                        (* send frame *)
                        fbSend(bExecute  := FALSE);
                        fbSend(sSrvNetID := '',
                               hSocket   := fbConnect.hSocket,
                               cbLen     := SIZEOF(toServer.Header) + _byteCount,(* size of header + size of user data *)
                               pSrc      := ADR(toServer),(* pointer to the frame data *)
                               bExecute  := TRUE,
                               tTimeout  := T#5s);

                        tx_state := 1;
                    END_IF
                1:(* wait until send not busy *)
                    fbSend( bExecute := FALSE );
                    IF NOT fbSend.bBusy THEN
                        tx_state := 0;
                        IF NOT fbSend.bError THEN(* no error *)
                            ;
                        ELSE(* send error => log error and disconnect *)
                            errors.Error(nErrId := fbSend.nErrId );
                            bDisconnect := TRUE;(* set flag *)
                        END_IF
                    END_IF
            END_CASE

            (* ------------------------------------------- Get/fetch rx data ----------------------------------------------------------------- *)
            CASE rx_state OF
                0:
                    IF NOT bDisconnect THEN
                        pollTimer( IN := TRUE );
                        IF pollTimer.Q THEN
                            pollTimer( IN := FALSE );

                            fbReceive( bExecute := FALSE );
                            fbReceive( 	sSrvNetId	:= '',
                            hSocket		:= fbConnect.hSocket,
                            cbLen		:= SIZEOF(fromServer) - cbReceived,
                            pDest		:= ADR(fromServer) + cbReceived,
                            bExecute	:= TRUE,
                            tTimeout	:= T#5s );
                            rx_state := 1;
                        END_IF
                    END_IF
                1:(* wait until receive not busy *)
                    fbReceive( bExecute := FALSE );
                    IF NOT fbReceive.bBusy THEN
                        rx_state := 0;
                        IF NOT fbReceive.bError THEN
                            IF fbReceive.nRecBytes > 0 THEN (* some bytes received *)

                                pollTimer( PT := T#0s );(* increase polling speed *)
                                cbReceived := cbReceived + fbReceive.nRecBytes;

                                (* parse received bytes *)
                                REPEAT
                                    bAbort := TRUE;(* set flag *)
                                    IF cbReceived >= SIZEOF(fromServer.Header) THEN (* all header bytes received => check header data *)

                                        (* correct header data *)
                                        fromServer.Header.ByteCount    := BE32_TO_HOST(fromServer.Header.ByteCount);
                                        Counter                        := fromServer.Header.Counter;
                                        fromServer.Header.SentTime     := BE32_TO_HOST(fromServer.Header.SentTime);
                                        fromServer.Header.DatagramType := BE32_TO_HOST(fromServer.Header.DatagramType);

                                        IF (fromServer.Header.ByteCount <= SIZEOF( fromServer.Payload))(* check frame (user data) length *)
                                        THEN

                                            cbRx := SIZEOF(fromServer.Header) + fromServer.Header.ByteCount;(* calculate the (expected) length of the rx frame *)
                                            IF cbReceived >= cbRx  THEN (* all frame bytes received? *)

                                               (* currently only use the data on a 32 Bit raw image *)
                                                IF fromServer.Header.DatagramType = MNG_Raw32BitImage THEN

                                                    IF 48 = (fromServer.Header.ByteCount - 4) THEN

                                                        (* BOOL Cocktail_Holder1_00_VACUUM *)
                                                        Inputs.Cocktail_Holder1_00_VACUUM := fromServer.Payload[2]<>0;

                                                        (* BOOL DetectionCookieAdapter1_00_IR *)
                                                        Inputs.DetectionCookieAdapter1_00_IR := fromServer.Payload[3]<>0;

                                                        (* BOOL Cocktail_Holder2_00_VACUUM *)
                                                        Inputs.Cocktail_Holder2_00_VACUUM := fromServer.Payload[4]<>0;

                                                        (* BOOL DetectionCookieAdapter2_00_IR *)
                                                        Inputs.DetectionCookieAdapter2_00_IR := fromServer.Payload[5]<>0;

                                                        (* BOOL Cocktail_Holder3_00_VACUUM *)
                                                        Inputs.Cocktail_Holder3_00_VACUUM := fromServer.Payload[6]<>0;

                                                        (* BOOL DetectionCookieAdapter3_00_IR *)
                                                        Inputs.DetectionCookieAdapter3_00_IR := fromServer.Payload[7]<>0;

                                                        (* BOOL Cocktail_Holder4_00_VACUUM *)
                                                        Inputs.Cocktail_Holder4_00_VACUUM := fromServer.Payload[8]<>0;

                                                        (* BOOL DetectionCookieAdapter4_00_IR *)
                                                        Inputs.DetectionCookieAdapter4_00_IR := fromServer.Payload[9]<>0;

                                                        (* BOOL Cocktail_Holder5_00_VACUUM *)
                                                        Inputs.Cocktail_Holder5_00_VACUUM := fromServer.Payload[10]<>0;

                                                        (* BOOL DetectionCookieAdapter5_00_IR *)
                                                        Inputs.DetectionCookieAdapter5_00_IR := fromServer.Payload[11]<>0;

                                                        (* BOOL Cocktail_Holder6_00_VACUUM *)
                                                        Inputs.Cocktail_Holder6_00_VACUUM := fromServer.Payload[12]<>0;

                                                        (* BOOL DetectionCookieAdapter6_00_IR *)
                                                        Inputs.DetectionCookieAdapter6_00_IR := fromServer.Payload[13]<>0;

                                                    ELSE(* receive error: invalid frame format/data *)
                                                        errors.Error(nErrId := PLCPRJ_ERROR_INVALID_IO_FORMAT_RECEIVED );
                                                    END_IF

                                                END_IF

                                                MEMMOVE( ADR( fromServer ), ADR( fromServer ) + cbRx,  cbReceived - cbRx );(* shift the remaining rx bytes *)
                                                cbReceived := cbReceived - cbRx;(* recalculate the size of the remaining rx bytes *)

                                                bAbort := FALSE;(* reset flag, try to parse next frame *)

                                                (* ELSE repeat reading *)
                                            END_IF

                                        ELSE(* receive error: invalid frame format/data *)
                                            errors.Error(nErrId := PLCPRJ_ERROR_INVALID_FRAME_FORMAT );
                                            bDisconnect := TRUE;(* set flag *)
                                        END_IF
                                        (* ELSE repeat reading *)
                                    END_IF (* IF cbReceived >= SIZEOF(rxFrame.head) THEN *)

                                UNTIL bAbort
                                END_REPEAT

                            ELSE(* fbReceive.nRecBytes = 0, repeat reading *)
                                pollTimer( PT := PLCPRJ_RECEIVER_POLLING_CYCLE_TIME );(* slow down the polling cycle *)
                            END_IF(* IF fbReceive.nRecBytes > 0 THEN *)
                        ELSE(* receive error => log error and disconnect *)
                            errors.Error(nErrId := fbReceive.nErrId );
                            bDisconnect := TRUE;(* set flag *)
                        END_IF

                    END_IF(*IF NOT fbReceive.bBusy THEN*)

            END_CASE

        END_IF

    3:(* disconnect *)
        fbConnect( bEnable:= FALSE, eState=>eState );
        IF eState = eSOCKET_DISCONNECTED THEN
            state := 0;
        END_IF

END_CASE

END_FUNCTION_BLOCK

// ---- POUs/industrialPhysics/FB_LogFifo.TcPOU
/// Log/debug/error message fifo 
FUNCTION_BLOCK FB_LogFifo
VAR_INPUT
	/// TRUE => Enable log message output, FALSE => Disable 
	bLog: BOOL := FALSE;
	/// Log message description string (allows the identification of log message source) 
	sPrefix: STRING := 'Unknown::';
	/// String message to add (write) to the fifo 
	sMessage: STRING := '';
	/// Error code to add (write) to the fifo 
	nErrID: UDINT := 0;
	/// Socket connection handle 
	hSocket: T_HSOCKET;
END_VAR
VAR_OUTPUT
	/// TRUE = New entry added or removed succesfully, FALSE = Fifo overflow or fifo empty 
	bOk: BOOL;
	/// String entry removed (read) from fifo 
	sGet: T_MaxString := '';
	/// Number of fifo entries 
	nCount: UDINT := 0;
END_VAR
VAR
	/// Basic (lower level) string buffer control function block 
	fbBuffer: FB_StringRingBuffer;
	/// Internal buffer memory 
	buffer: ARRAY[0..PLCPRJ_BUFFER_SIZE] OF BYTE;
	sSource: T_MaxString;
	sPut: T_MaxString;
END_VAR

;

ACTION Remove:
(* Removes oldest fifo entry *)
IF nCount = 0 THEN
	sGet := '';
	bOk := FALSE;
	RETURN;
END_IF

fbBuffer.A_RemoveHead( pBuffer:= ADR(buffer), cbBuffer:= SIZEOF(buffer),
						getValue=>sGet, bOk=>bOk, nCount=>nCount );
END_ACTION

ACTION Message:
(* Adds new fifo entry *)
sPut := CONCAT( CONCAT( sPrefix, sMessage ), CONCAT( '::', HSOCKET_TO_STRING(hSocket) ) );
fbBuffer.A_AddTail( pBuffer:= ADR(buffer), cbBuffer:= SIZEOF(buffer),
					putValue:= sPut, bOk=>bOk, nCount=>nCount );
IF bOk THEN
	IF bLog THEN(* Log information message *)
		ADSLOGSTR( ADSLOG_MSGTYPE_HINT OR ADSLOG_MSGTYPE_LOG, '%s', sPut );	
	END_IF
END_IF
END_ACTION

ACTION Clear:
(* Clears all fifo entries *)
fbBuffer.A_Reset( 	pBuffer := ADR( buffer ), cbBuffer := SIZEOF( buffer ), 
					bOk=>bOk, nCount=>nCount, getValue=>sGet );
END_ACTION

ACTION Error:
(* Adds new fifo entry *)
IF nErrID = 0 THEN
	sSource := '::Error: 0x';
ELSIF ( nErrID AND 16#80000000) = 16#80000000 THEN
	IF nErrID = 16#80072746 THEN
		sSource := '::Win32 error (the connection is reset by remote side): 0x';
	ELSE
		sSource := '::Win32 error: 0x';
	END_IF
ELSIF (nErrID AND 16#00008100) = 16#00008100 THEN
	CASE nErrID OF
		PLCPRJ_ERROR_RECEIVE_TIMEOUT:
			sSource := '::PLC sample project receive timeout error: 0x';
		PLCPRJ_ERROR_SENDFIFO_OVERFLOW:
			sSource := '::PLC sample project send fifo overflow error: 0x';
		PLCPRJ_ERROR_RECFIFO_OVERFLOW:
			sSource := '::PLC sample project receive fifo overflow error: 0x';
		PLCPRJ_ERROR_INVALID_FRAME_FORMAT:
			sSource := '::PLC sample project invalid frame format error: 0x';
	ELSE
		sSource := '::Other PLC sample project error: 0x';
	END_CASE
ELSIF (nErrID AND 16#00008000) = 16#00008000 THEN
	sSource := '::Internal TCP/IP Connection Server error: 0x';
ELSE
	sSource := '::TwinCAT System error: 0x';
END_IF

sPut := CONCAT( CONCAT( CONCAT( sPrefix, sMessage ), sSource ), DWORD_TO_HEXSTR( nErrID AND 16#FFFF, 0, FALSE ) ); 

fbBuffer.A_AddTail( pBuffer:= ADR(buffer), cbBuffer:= SIZEOF(buffer),
					putValue:= sPut, bOk=>bOk, nCount=>nCount );
IF bOk THEN
	IF bLog THEN(* Log error message *)
		ADSLOGSTR( ADSLOG_MSGTYPE_ERROR OR ADSLOG_MSGTYPE_LOG, '%s', sPut );	
	END_IF
END_IF
END_ACTION

END_FUNCTION_BLOCK

// ---- POUs/industrialPhysics/FB_IOLink.TcPOU
FUNCTION_BLOCK FB_IOLink
VAR_INPUT
	goon : BOOL  := TRUE;
	inputs: MNG_Application_Inputs_32Bit;
	
	
END_VAR
VAR_OUTPUT
	outputs: MNG_Application_Outputs_32Bit;
END_VAR
VAR
	timer: ARRAY[1..6] OF Tc2_Standard.TON;
	state: ARRAY[1..6] OF INT := [0, 0, 0, 0, 0, 0];
	deltaMover: ARRAY[1..6] OF LREAL;
END_VAR

// Application code follows here:

IF goon THEN

outputs.Fahrachse1_00_ChainDrvActual := GVL.ax[1].NcToPlc.SetPos/1000;
outputs.Fahrachse2_00_ChainDrvActual := GVL.ax[2].NcToPlc.SetPos/1000;
outputs.Fahrachse3_00_ChainDrvActual := GVL.ax[3].NcToPlc.SetPos/1000;
outputs.Fahrachse4_00_ChainDrvActual := GVL.ax[4].NcToPlc.SetPos/1000;
outputs.Fahrachse5_00_ChainDrvActual := GVL.ax[5].NcToPlc.SetPos/1000;
outputs.Fahrachse6_00_ChainDrvActual := GVL.ax[6].NcToPlc.SetPos/1000;


outputs.LED_0_00_00_on1 := GVL.LampInterface[1][1];
outputs.LED_0_05_00_on1 := GVL.LampInterface[1][2];
outputs.LED_0_10_00_on1 := GVL.LampInterface[1][3];
outputs.LED_0_15_00_on1 := GVL.LampInterface[1][4];
outputs.LED_0_20_00_on1 := GVL.LampInterface[1][5];
outputs.LED_0_25_00_on1 := GVL.LampInterface[1][6];
outputs.LED_0_30_00_on1 := GVL.LampInterface[1][7];
outputs.LED_0_35_00_on1 := GVL.LampInterface[1][8];
outputs.LED_0_40_00_on1 := GVL.LampInterface[1][9];
outputs.LED_0_45_00_on1 := GVL.LampInterface[1][10];
outputs.LED_0_50_00_on1 := GVL.LampInterface[1][11];
outputs.LED_0_55_00_on1 := GVL.LampInterface[1][12];
outputs.LED_0_60_00_on1 := GVL.LampInterface[1][13];
outputs.LED_0_65_00_on1 := GVL.LampInterface[1][14];
outputs.LED_0_70_00_on1 := GVL.LampInterface[1][15];
outputs.LED_0_75_00_on1 := GVL.LampInterface[1][16];
outputs.LED_0_80_00_on1 := GVL.LampInterface[1][17];
outputs.LED_0_85_00_on1 := GVL.LampInterface[1][18];
outputs.LED_0_90_00_on1 := GVL.LampInterface[1][19];
outputs.LED_0_95_00_on1 := GVL.LampInterface[1][20];
outputs.LED_1_00_00_on1 := GVL.LampInterface[1][21];
outputs.LED_1_05_00_on1 := GVL.LampInterface[1][22];
outputs.LED_1_10_00_on1 := GVL.LampInterface[1][23];
outputs.LED_1_15_00_on1 := GVL.LampInterface[1][24];
outputs.LED_1_20_00_on1 := GVL.LampInterface[1][25];
outputs.LED_1_25_00_on1 := GVL.LampInterface[1][26];
outputs.LED_1_30_00_on1 := GVL.LampInterface[1][27];
outputs.LED_1_35_00_on1 := GVL.LampInterface[1][28];
outputs.LED_1_40_00_on1 := GVL.LampInterface[1][29];
outputs.LED_1_45_00_on1 := GVL.LampInterface[1][30];
(*
outputs.LED_1_50_00_on1 := GVL.LampInterface[1][31];
outputs.LED_1_55_00_on1 := GVL.LampInterface[1][32];
outputs.LED_1_60_00_on1 := GVL.LampInterface[1][33];
outputs.LED_1_65_00_on1 := GVL.LampInterface[1][34];
outputs.LED_1_70_00_on1 := GVL.LampInterface[1][35];
outputs.LED_1_75_00_on1 := GVL.LampInterface[1][36];
outputs.LED_1_80_00_on1 := GVL.LampInterface[1][37];
outputs.LED_1_85_00_on1 := GVL.LampInterface[1][38];
outputs.LED_1_90_00_on1 := GVL.LampInterface[1][39];
outputs.LED_1_95_00_on1 := GVL.LampInterface[1][40];
*)
outputs.LED_2_00_00_on1 := GVL.LampInterface[1][41];
outputs.LED_2_05_00_on1 := GVL.LampInterface[1][42];
outputs.LED_2_10_00_on1 := GVL.LampInterface[1][43];
outputs.LED_2_15_00_on1 := GVL.LampInterface[1][44];
outputs.LED_2_20_00_on1 := GVL.LampInterface[1][45];
outputs.LED_2_25_00_on1 := GVL.LampInterface[1][46];
outputs.LED_2_30_00_on1 := GVL.LampInterface[1][47];
outputs.LED_2_35_00_on1 := GVL.LampInterface[1][48];
outputs.LED_2_40_00_on1 := GVL.LampInterface[1][49];
outputs.LED_2_45_00_on1 := GVL.LampInterface[1][50];
outputs.LED_2_50_00_on1 := GVL.LampInterface[1][51];
outputs.LED_2_55_00_on1 := GVL.LampInterface[1][52];
outputs.LED_2_60_00_on1 := GVL.LampInterface[1][53];
outputs.LED_2_65_00_on1 := GVL.LampInterface[1][54];
outputs.LED_2_70_00_on1 := GVL.LampInterface[1][55];
outputs.LED_2_75_00_on1 := GVL.LampInterface[1][56];
outputs.LED_2_80_00_on1 := GVL.LampInterface[1][57];
outputs.LED_2_85_00_on1 := GVL.LampInterface[1][58];
outputs.LED_2_90_00_on1 := GVL.LampInterface[1][59];
outputs.LED_2_95_00_on1 := GVL.LampInterface[1][60];
outputs.LED_3_00_00_on1 := GVL.LampInterface[1][61];
outputs.LED_3_05_00_on1 := GVL.LampInterface[1][62];
outputs.LED_3_10_00_on1 := GVL.LampInterface[1][63];
outputs.LED_3_15_00_on1 := GVL.LampInterface[1][64];
outputs.LED_3_20_00_on1 := GVL.LampInterface[1][65];
outputs.LED_3_25_00_on1 := GVL.LampInterface[1][66];
outputs.LED_3_30_00_on1 := GVL.LampInterface[1][67];
outputs.LED_3_35_00_on1 := GVL.LampInterface[1][68];
outputs.LED_3_40_00_on1 := GVL.LampInterface[1][69];
outputs.LED_3_45_00_on1 := GVL.LampInterface[1][70];
(*
outputs.LED_3_50_00_on1 := GVL.LampInterface[1][71];
outputs.LED_3_55_00_on1 := GVL.LampInterface[1][72];
outputs.LED_3_60_00_on1 := GVL.LampInterface[1][73];
outputs.LED_3_65_00_on1 := GVL.LampInterface[1][74];
outputs.LED_3_70_00_on1 := GVL.LampInterface[1][75];
outputs.LED_3_75_00_on1 := GVL.LampInterface[1][76];
outputs.LED_3_80_00_on1 := GVL.LampInterface[1][77];
outputs.LED_3_85_00_on1 := GVL.LampInterface[1][78];
outputs.LED_3_90_00_on1 := GVL.LampInterface[1][79];
outputs.LED_3_95_00_on1 := GVL.LampInterface[1][80];
*)

// Lampe 2:

outputs.LED_0_00_00_on2 := GVL.LampInterface[2][1];;
outputs.LED_0_05_00_on2 := GVL.LampInterface[2][2];;
outputs.LED_0_10_00_on2 := GVL.LampInterface[2][3];;
outputs.LED_0_15_00_on2 := GVL.LampInterface[2][4];;
outputs.LED_0_20_00_on2 := GVL.LampInterface[2][5];;
outputs.LED_0_25_00_on2 := GVL.LampInterface[2][6];;
outputs.LED_0_30_00_on2 := GVL.LampInterface[2][7];;
outputs.LED_0_35_00_on2 := GVL.LampInterface[2][8];;
outputs.LED_0_40_00_on2 := GVL.LampInterface[2][9];;
outputs.LED_0_45_00_on2 := GVL.LampInterface[2][10];
outputs.LED_0_50_00_on2 := GVL.LampInterface[2][11];
outputs.LED_0_55_00_on2 := GVL.LampInterface[2][12];
outputs.LED_0_60_00_on2 := GVL.LampInterface[2][13];
outputs.LED_0_65_00_on2 := GVL.LampInterface[2][14];
outputs.LED_0_70_00_on2 := GVL.LampInterface[2][15];
outputs.LED_0_75_00_on2 := GVL.LampInterface[2][16];
outputs.LED_0_80_00_on2 := GVL.LampInterface[2][17];
outputs.LED_0_85_00_on2 := GVL.LampInterface[2][18];
outputs.LED_0_90_00_on2 := GVL.LampInterface[2][19];
outputs.LED_0_95_00_on2 := GVL.LampInterface[2][20];
outputs.LED_1_00_00_on2 := GVL.LampInterface[2][21];
outputs.LED_1_05_00_on2 := GVL.LampInterface[2][22];
outputs.LED_1_10_00_on2 := GVL.LampInterface[2][23];
outputs.LED_1_15_00_on2 := GVL.LampInterface[2][24];
outputs.LED_1_20_00_on2 := GVL.LampInterface[2][25];
outputs.LED_1_25_00_on2 := GVL.LampInterface[2][26];
outputs.LED_1_30_00_on2 := GVL.LampInterface[2][27];
outputs.LED_1_35_00_on2 := GVL.LampInterface[2][28];
outputs.LED_1_40_00_on2 := GVL.LampInterface[2][29];
outputs.LED_1_45_00_on2 := GVL.LampInterface[2][30];
(*                                                 
outputs.LED_1_50_00_on2 := GVL.LampInterface[2][31];
outputs.LED_1_55_00_on2 := GVL.LampInterface[2][32];
outputs.LED_1_60_00_on2 := GVL.LampInterface[2][33];
outputs.LED_1_65_00_on2 := GVL.LampInterface[2][34];
outputs.LED_1_70_00_on2 := GVL.LampInterface[2][35];
outputs.LED_1_75_00_on2 := GVL.LampInterface[2][36];
outputs.LED_1_80_00_on2 := GVL.LampInterface[2][37];
outputs.LED_1_85_00_on2 := GVL.LampInterface[2][38];
outputs.LED_1_90_00_on2 := GVL.LampInterface[2][39];
outputs.LED_1_95_00_on2 := GVL.LampInterface[2][40];
*)                                                 
outputs.LED_2_00_00_on2 := GVL.LampInterface[2][41];
outputs.LED_2_05_00_on2 := GVL.LampInterface[2][42];
outputs.LED_2_10_00_on2 := GVL.LampInterface[2][43];
outputs.LED_2_15_00_on2 := GVL.LampInterface[2][44];
outputs.LED_2_20_00_on2 := GVL.LampInterface[2][45];
outputs.LED_2_25_00_on2 := GVL.LampInterface[2][46];
outputs.LED_2_30_00_on2 := GVL.LampInterface[2][47];
outputs.LED_2_35_00_on2 := GVL.LampInterface[2][48];
outputs.LED_2_40_00_on2 := GVL.LampInterface[2][49];
outputs.LED_2_45_00_on2 := GVL.LampInterface[2][50];
outputs.LED_2_50_00_on2 := GVL.LampInterface[2][51];
outputs.LED_2_55_00_on2 := GVL.LampInterface[2][52];
outputs.LED_2_60_00_on2 := GVL.LampInterface[2][53];
outputs.LED_2_65_00_on2 := GVL.LampInterface[2][54];
outputs.LED_2_70_00_on2 := GVL.LampInterface[2][55];
outputs.LED_2_75_00_on2 := GVL.LampInterface[2][56];
outputs.LED_2_80_00_on2 := GVL.LampInterface[2][57];
outputs.LED_2_85_00_on2 := GVL.LampInterface[2][58];
outputs.LED_2_90_00_on2 := GVL.LampInterface[2][59];
outputs.LED_2_95_00_on2 := GVL.LampInterface[2][60];
outputs.LED_3_00_00_on2 := GVL.LampInterface[2][61];
outputs.LED_3_05_00_on2 := GVL.LampInterface[2][62];
outputs.LED_3_10_00_on2 := GVL.LampInterface[2][63];
outputs.LED_3_15_00_on2 := GVL.LampInterface[2][64];
outputs.LED_3_20_00_on2 := GVL.LampInterface[2][65];
outputs.LED_3_25_00_on2 := GVL.LampInterface[2][66];
outputs.LED_3_30_00_on2 := GVL.LampInterface[2][67];
outputs.LED_3_35_00_on2 := GVL.LampInterface[2][68];
outputs.LED_3_40_00_on2 := GVL.LampInterface[2][69];
outputs.LED_3_45_00_on2 := GVL.LampInterface[2][70];
(*                                                 
outputs.LED_3_50_00_on2 := GVL.LampInterface[2][71];
outputs.LED_3_55_00_on2 := GVL.LampInterface[2][72];
outputs.LED_3_60_00_on2 := GVL.LampInterface[2][73];
outputs.LED_3_65_00_on2 := GVL.LampInterface[2][74];
outputs.LED_3_70_00_on2 := GVL.LampInterface[2][75];
outputs.LED_3_75_00_on2 := GVL.LampInterface[2][76];
outputs.LED_3_80_00_on2 := GVL.LampInterface[2][77];
outputs.LED_3_85_00_on2 := GVL.LampInterface[2][78];
outputs.LED_3_90_00_on2 := GVL.LampInterface[2][79];
outputs.LED_3_95_00_on2 := GVL.LampInterface[2][80];
*)

// Lampe 3:

outputs.LED_0_00_00_on3 := GVL.LampInterface[3][1];;
outputs.LED_0_05_00_on3 := GVL.LampInterface[3][2];;
outputs.LED_0_10_00_on3 := GVL.LampInterface[3][3];;
outputs.LED_0_15_00_on3 := GVL.LampInterface[3][4];;
outputs.LED_0_20_00_on3 := GVL.LampInterface[3][5];;
outputs.LED_0_25_00_on3 := GVL.LampInterface[3][6];;
outputs.LED_0_30_00_on3 := GVL.LampInterface[3][7];;
outputs.LED_0_35_00_on3 := GVL.LampInterface[3][8];;
outputs.LED_0_40_00_on3 := GVL.LampInterface[3][9];;
outputs.LED_0_45_00_on3 := GVL.LampInterface[3][10];
outputs.LED_0_50_00_on3 := GVL.LampInterface[3][11];
outputs.LED_0_55_00_on3 := GVL.LampInterface[3][12];
outputs.LED_0_60_00_on3 := GVL.LampInterface[3][13];
outputs.LED_0_65_00_on3 := GVL.LampInterface[3][14];
outputs.LED_0_70_00_on3 := GVL.LampInterface[3][15];
outputs.LED_0_75_00_on3 := GVL.LampInterface[3][16];
outputs.LED_0_80_00_on3 := GVL.LampInterface[3][17];
outputs.LED_0_85_00_on3 := GVL.LampInterface[3][18];
outputs.LED_0_90_00_on3 := GVL.LampInterface[3][19];
outputs.LED_0_95_00_on3 := GVL.LampInterface[3][20];
outputs.LED_1_00_00_on3 := GVL.LampInterface[3][21];
outputs.LED_1_05_00_on3 := GVL.LampInterface[3][22];
outputs.LED_1_10_00_on3 := GVL.LampInterface[3][23];
outputs.LED_1_15_00_on3 := GVL.LampInterface[3][24];
outputs.LED_1_20_00_on3 := GVL.LampInterface[3][25];
outputs.LED_1_25_00_on3 := GVL.LampInterface[3][26];
outputs.LED_1_30_00_on3 := GVL.LampInterface[3][27];
outputs.LED_1_35_00_on3 := GVL.LampInterface[3][28];
outputs.LED_1_40_00_on3 := GVL.LampInterface[3][29];
outputs.LED_1_45_00_on3 := GVL.LampInterface[3][30];
(*                                                 
outputs.LED_1_50_00_on3 := GVL.LampInterface[3][31];
outputs.LED_1_55_00_on3 := GVL.LampInterface[3][32];
outputs.LED_1_60_00_on3 := GVL.LampInterface[3][33];
outputs.LED_1_65_00_on3 := GVL.LampInterface[3][34];
outputs.LED_1_70_00_on3 := GVL.LampInterface[3][35];
outputs.LED_1_75_00_on3 := GVL.LampInterface[3][36];
outputs.LED_1_80_00_on3 := GVL.LampInterface[3][37];
outputs.LED_1_85_00_on3 := GVL.LampInterface[3][38];
outputs.LED_1_90_00_on3 := GVL.LampInterface[3][39];
outputs.LED_1_95_00_on3 := GVL.LampInterface[3][40];
*)                                                 
outputs.LED_2_00_00_on3 := GVL.LampInterface[3][41];
outputs.LED_2_05_00_on3 := GVL.LampInterface[3][42];
outputs.LED_2_10_00_on3 := GVL.LampInterface[3][43];
outputs.LED_2_15_00_on3 := GVL.LampInterface[3][44];
outputs.LED_2_20_00_on3 := GVL.LampInterface[3][45];
outputs.LED_2_25_00_on3 := GVL.LampInterface[3][46];
outputs.LED_2_30_00_on3 := GVL.LampInterface[3][47];
outputs.LED_2_35_00_on3 := GVL.LampInterface[3][48];
outputs.LED_2_40_00_on3 := GVL.LampInterface[3][49];
outputs.LED_2_45_00_on3 := GVL.LampInterface[3][50];
outputs.LED_2_50_00_on3 := GVL.LampInterface[3][51];
outputs.LED_2_55_00_on3 := GVL.LampInterface[3][52];
outputs.LED_2_60_00_on3 := GVL.LampInterface[3][53];
outputs.LED_2_65_00_on3 := GVL.LampInterface[3][54];
outputs.LED_2_70_00_on3 := GVL.LampInterface[3][55];
outputs.LED_2_75_00_on3 := GVL.LampInterface[3][56];
outputs.LED_2_80_00_on3 := GVL.LampInterface[3][57];
outputs.LED_2_85_00_on3 := GVL.LampInterface[3][58];
outputs.LED_2_90_00_on3 := GVL.LampInterface[3][59];
outputs.LED_2_95_00_on3 := GVL.LampInterface[3][60];
outputs.LED_3_00_00_on3 := GVL.LampInterface[3][61];
outputs.LED_3_05_00_on3 := GVL.LampInterface[3][62];
outputs.LED_3_10_00_on3 := GVL.LampInterface[3][63];
outputs.LED_3_15_00_on3 := GVL.LampInterface[3][64];
outputs.LED_3_20_00_on3 := GVL.LampInterface[3][65];
outputs.LED_3_25_00_on3 := GVL.LampInterface[3][66];
outputs.LED_3_30_00_on3 := GVL.LampInterface[3][67];
outputs.LED_3_35_00_on3 := GVL.LampInterface[3][68];
outputs.LED_3_40_00_on3 := GVL.LampInterface[3][69];
outputs.LED_3_45_00_on3 := GVL.LampInterface[3][70];
(*                                                 
outputs.LED_3_50_00_on3 := GVL.LampInterface[3][71];
outputs.LED_3_55_00_on3 := GVL.LampInterface[3][72];
outputs.LED_3_60_00_on3 := GVL.LampInterface[3][73];
outputs.LED_3_65_00_on3 := GVL.LampInterface[3][74];
outputs.LED_3_70_00_on3 := GVL.LampInterface[3][75];
outputs.LED_3_75_00_on3 := GVL.LampInterface[3][76];
outputs.LED_3_80_00_on3 := GVL.LampInterface[3][77];
outputs.LED_3_85_00_on3 := GVL.LampInterface[3][78];
outputs.LED_3_90_00_on3 := GVL.LampInterface[3][79];
outputs.LED_3_95_00_on3 := GVL.LampInterface[3][80];
*)


END_IF


CASE state[1] OF
	0: IF inputs.DetectionCookieAdapter1_00_IR THEN
			state[1] := 10;
	   END_IF
	   outputs.Cocktail_Holder1_00_GRIP := FALSE;
	10:
		timer[1].PT := INT_TO_TIME(5000) ;
		timer[1](IN := FALSE);
		timer[1](IN := TRUE);
		state[1] := 20;
	20:
		timer[1]();
		IF timer[1].Q THEN
			outputs.Cocktail_Holder1_00_GRIP := TRUE;
		END_IF
				
END_CASE

CASE state[2] OF
	0: IF inputs.DetectionCookieAdapter2_00_IR THEN
			state[2] := 10;
	   END_IF
	   outputs.Cocktail_Holder2_00_GRIP := FALSE;
	10:
		timer[2].PT := INT_TO_TIME(5000) ;
		timer[2](IN := FALSE);
		timer[2](IN := TRUE);
		state[2] := 20;
	20:
		timer[2]();
		IF timer[2].Q THEN
			outputs.Cocktail_Holder2_00_GRIP := TRUE;
		END_IF
				
END_CASE

CASE state[3] OF
	0: IF inputs.DetectionCookieAdapter3_00_IR THEN
			state[3] := 10;
	   END_IF
	   outputs.Cocktail_Holder3_00_GRIP := FALSE;
	10:
		timer[3].PT := INT_TO_TIME(5000) ;
		timer[3](IN := FALSE);
		timer[3](IN := TRUE);
		state[3] := 20;
	20:
		timer[3]();
		IF timer[3].Q THEN
			outputs.Cocktail_Holder3_00_GRIP := TRUE;
		END_IF
				
END_CASE

CASE state[4] OF
	0: IF inputs.DetectionCookieAdapter4_00_IR THEN
			state[4] := 10;
	   END_IF
	   outputs.Cocktail_Holder4_00_GRIP := FALSE;
	10:
		timer[4].PT := INT_TO_TIME(5000) ;
		timer[4](IN := FALSE);
		timer[4](IN := TRUE);
		state[4] := 20;
	20:
		timer[4]();
		IF timer[4].Q THEN
			outputs.Cocktail_Holder4_00_GRIP := TRUE;
		END_IF
END_CASE
		
CASE state[5] OF
	0: IF inputs.DetectionCookieAdapter5_00_IR THEN
			state[5] := 10;
	   END_IF
	   outputs.Cocktail_Holder5_00_GRIP := FALSE;
	10:
		timer[5].PT := INT_TO_TIME(5000) ;
		timer[5](IN := FALSE);
		timer[5](IN := TRUE);
		state[5] := 20;
	20:
		timer[5]();
		IF timer[5].Q THEN
			outputs.Cocktail_Holder5_00_GRIP := TRUE;
		END_IF
				
END_CASE

CASE state[6] OF
	0: IF inputs.DetectionCookieAdapter6_00_IR THEN
			state[6] := 10;
	   END_IF
	   outputs.Cocktail_Holder6_00_GRIP := FALSE;
	10:
		timer[6].PT := INT_TO_TIME(5000) ;
		timer[6](IN := FALSE);
		timer[6](IN := TRUE);
		state[6] := 20;
	20:
		timer[6]();
		IF timer[6].Q THEN
			outputs.Cocktail_Holder6_00_GRIP := TRUE;
		END_IF
				
END_CASE

deltaMover[6] := GVL.ax[6].NcToPlc.SetPos/10-GVL.ax[5].NcToPlc.SetPos/10;
outputs.Cocktail_Holder_6_00_ACT_POS := 0.32 - 0.02667*deltaMover[6];
IF deltaMover[6] > 12 THEN
	outputs.Cocktail_Holder_6_00_ACT_POS := 0;
END_IF

deltaMover[5] := GVL.ax[5].NcToPlc.SetPos/10-GVL.ax[4].NcToPlc.SetPos/10;
outputs.Cocktail_Holder_5_00_ACT_POS := 0.32 - 0.02667*deltaMover[5];
IF deltaMover[5] > 12 THEN
	outputs.Cocktail_Holder_5_00_ACT_POS := 0;
END_IF

deltaMover[4] := GVL.ax[4].NcToPlc.SetPos/10-GVL.ax[3].NcToPlc.SetPos/10;
outputs.Cocktail_Holder_4_00_ACT_POS := 0.32 - 0.02667*deltaMover[4];
IF deltaMover[4] > 12 THEN
	outputs.Cocktail_Holder_4_00_ACT_POS := 0;
END_IF

deltaMover[3] := GVL.ax[3].NcToPlc.SetPos/10-GVL.ax[2].NcToPlc.SetPos/10;
outputs.Cocktail_Holder_3_00_ACT_POS := 0.32 - 0.02667*deltaMover[3];
IF deltaMover[3] > 12 THEN
	outputs.Cocktail_Holder_3_00_ACT_POS := 0;
END_IF

deltaMover[2] := GVL.ax[2].NcToPlc.SetPos/10-GVL.ax[1].NcToPlc.SetPos/10;
outputs.Cocktail_Holder_2_00_ACT_POS := 0.32 - 0.02667*deltaMover[2];
IF deltaMover[2] > 12 THEN
	outputs.Cocktail_Holder_2_00_ACT_POS := 0;
END_IF

deltaMover[1] := GVL.ax[1].NcToPlc.SetPos/10-GVL.ax[6].NcToPlc.SetPos/10+400;
outputs.Cocktail_Holder_1_00_ACT_POS := 0.32 - 0.02667*deltaMover[1];
IF deltaMover[1] > 12 THEN
	outputs.Cocktail_Holder_1_00_ACT_POS := 0;
END_IF
// Moverpaar 1:
//linke hälfte
outputs.Seitenwand_00_reserved_colour02 := MoverInfo[1].reserved;
outputs.Seitenwand_00_blocked_colour02	:= MoverInfo[1].blocked;
outputs.Seitenwand_00_error_colour02	:= MoverInfo[1].surpressed;
outputs.Seitenwand_00_reserved_colour02 := MoverInfo[1].reserved;
outputs.Seitenwand_00_blocked_colour02	:= MoverInfo[1].blocked;
//surpressed nur auf der einen seite ** outputs.Seitenwand_00_error_colour02	:= MoverInfo[1].surpressed;
//rechte hälfte
outputs.Seitenwand0_00_reserved_colour02 := MoverInfo[1].reserved;
outputs.Seitenwand0_00_blocked_colour02	:= MoverInfo[1].blocked;
outputs.Seitenwand0_00_error_colour02	:= MoverInfo[1].surpressed;
outputs.Seitenwand0_00_reserved_colour02 := MoverInfo[1].reserved;
outputs.Seitenwand0_00_blocked_colour02	:= MoverInfo[1].blocked;
outputs.Seitenwand0_00_error_colour02	:= MoverInfo[1].surpressed;

//moverpaar 2:

//linke hälfte
outputs.Seitenwand_00_reserved_colour04 := MoverInfo[2].reserved;
outputs.Seitenwand_00_blocked_colour04	:= MoverInfo[2].blocked;
outputs.Seitenwand_00_error_colour04	:= MoverInfo[2].surpressed;
outputs.Seitenwand_00_reserved_colour04 := MoverInfo[2].reserved;
outputs.Seitenwand_00_blocked_colour04	:= MoverInfo[2].blocked;
//surpressed nur auf der einen seite ** outputs.Seitenwand_00_error_colour02	:= MoverInfo[2].surpressed;
//rechte hälfte
outputs.Seitenwand0_00_reserved_colour04 := MoverInfo[2].reserved;
outputs.Seitenwand0_00_blocked_colour04	:= MoverInfo[2].blocked;
outputs.Seitenwand0_00_error_colour04	:= MoverInfo[2].surpressed;
outputs.Seitenwand0_00_reserved_colour04 := MoverInfo[2].reserved;
outputs.Seitenwand0_00_blocked_colour04	:= MoverInfo[2].blocked;
outputs.Seitenwand0_00_error_colour04	:= MoverInfo[2].surpressed;

//moverpaar 3:

//linke hälfte
outputs.Seitenwand_00_reserved_colour06 := MoverInfo[3].reserved;
outputs.Seitenwand_00_blocked_colour06	:= MoverInfo[3].blocked;
outputs.Seitenwand_00_error_colour06	:= MoverInfo[3].surpressed;
outputs.Seitenwand_00_reserved_colour06 := MoverInfo[3].reserved;
outputs.Seitenwand_00_blocked_colour06	:= MoverInfo[3].blocked;
//surpressed nur auf der einen seite ** outputs.Seitenwand_00_error_colour02	:= MoverInfo[3].surpressed;
//rechte hälfte
outputs.Seitenwand0_00_reserved_colour06 := MoverInfo[3].reserved;
outputs.Seitenwand0_00_blocked_colour06	:= MoverInfo[3].blocked;
outputs.Seitenwand0_00_error_colour06	:= MoverInfo[3].surpressed;
outputs.Seitenwand0_00_reserved_colour06 := MoverInfo[3].reserved;
outputs.Seitenwand0_00_blocked_colour06	:= MoverInfo[3].blocked;
outputs.Seitenwand0_00_error_colour06	:= MoverInfo[3].surpressed;

END_FUNCTION_BLOCK

// ---- POUs/CAHandle/MC2Handle/F_CurveSpeed.TcPOU
FUNCTION F_CurveSpeed : LREAL
VAR_INPUT
END_VAR
VAR
END_VAR

END_FUNCTION

// ---- POUs/CAHandle/MC2Handle/F_MoverInCurve.TcPOU
FUNCTION F_MoverInCurve : BOOL
VAR_INPUT
	Position: LREAL;
END_VAR
VAR
	pre1: LREAL := 1250.0;
	pre2: LREAL := 2250.0;
	end1: LREAL := 3250.0;
	end2: LREAL := 250.0;
END_VAR

F_MoverInCurve := F_CheckIfInSection(Position := Position, postposition := end1, preposition := pre1) or F_CheckIfInSection(Position := Position, postposition := end2, preposition := pre2);

END_FUNCTION

// ---- POUs/OPC Client/FB_OpcUaHandle.TcPOU
FUNCTION_BLOCK FB_OpcUaHandle
VAR_INPUT
	execute	: BOOL;
END_VAR
VAR_OUTPUT
	established	: BOOL;
	error		: BOOL;
END_VAR
VAR
	fbOpcUaHandle	: ARRAY [1..grpcnt] OF FB_Update;
	
	initdone	: BOOL := FALSE;
	i: INT;
END_VAR

IF execute THEN
	

		IF initdone THEN
				FOR i := 1 TO grpcnt DO
					fbOpcUaHandle[i](			
					Execute:= TRUE, 
					ModuleOutput:= Module[i].Output, 
					ModuleInput=> Module[i].Input, 
					established=> established, 
					error=> error);
				END_FOR
				
		ELSE
			fbOpcUaHandle[1](
					ServerUrl:= 'opc.tcp://192.168.175.230:4840', 
					NamespaceUri:= 'PLC1', 
					ClientName:= 'XTS1', 
					IdentifierInput:= 'GVL.OPCModule[1].Input', 
					IdentifierOutput:= 'GVL.OPCModule[1].Output', 
					Execute:= FALSE 
					);
			fbOpcUaHandle[2](
					ServerUrl:= 'opc.tcp://192.168.175.230:4840', 
					NamespaceUri:= 'PLC1', 
					ClientName:= 'XTS2', 
					IdentifierInput:= 'GVL.OPCModule[2].Input', 
					IdentifierOutput:= 'GVL.OPCModule[2].Output', 
					Execute:= FALSE 
					);
			fbOpcUaHandle[3](
					ServerUrl:= 'opc.tcp://192.168.175.230:4840', 
					NamespaceUri:= 'PLC1', 
					ClientName:= 'XTS3', 
					IdentifierInput:= 'GVL.OPCModule[3].Input', 
					IdentifierOutput:= 'GVL.OPCModule[3].Output', 
					Execute:= FALSE 
					);
			initdone := TRUE;
			
		
		
		END_IF
END_IF

END_FUNCTION_BLOCK

// ---- POUs/OPC Client/FB_Update.TcPOU
FUNCTION_BLOCK FB_Update
VAR_INPUT
	ServerUrl: STRING;
	NamespaceUri: STRING;
	ClientName: STRING;
	IdentifierInput: STRING;
	IdentifierOutput: STRING;
	Execute: BOOL;
	ModuleOutput: DUT_MODULE_INTERFACE_OUTPUT;
END_VAR
VAR_OUTPUT
	ModuleInput: DUT_MODULE_INTERFACE_INPUT;
	established	: BOOL;
	error		: BOOL;
END_VAR
VAR
	readestablished : BOOL;
	writeestablished : BOOL;
	fbConnect: FB_OPCServerConnect;
	fbRead: FB_ReadVariableOnce;
	fbWrite: FB_WriteVariableOnce;
	NamespaceIndex: UINT;
	ConnectionHdl: DWORD;
	state: INT;
END_VAR

IF Execute THEN	
error := FALSE;
established := FALSE;
CASE state OF
	
	0: state := 1;
	1: fbConnect(
			ServerUrl:= ServerUrl, 
			NamespaceUri:= NamespaceUri , 
			ClientName:= ClientName , 
			execute:= TRUE, 
			ConnectHdl=> ConnectionHdl , 
			Namespaceindex=> NamespaceIndex , 
			busy=> , 
			done=> , 
			error=> );
		IF fbConnect.done THEN
		state := 2;
		END_IF
		
		
		
	
	2: fbRead(
			IdentifierInput:= IdentifierInput, 
			NamespaceIndex:= NamespaceIndex, 
			ConnectionHdl:= ConnectionHdl, 
			execute:= TRUE, 
			ModuleInput=> ModuleInput, 
			done=> , 
			busy=> , 
			error=> );
		IF fbRead.done THEN
			readestablished := TRUE;
		END_IF
		state := 3;

			
	3:fbWrite(
		IdentifierOutput:= IdentifierOutput, 
		NamespaceIndex:= NamespaceIndex, 
		ConnectionHdl:= ConnectionHdl, 
		execute:= TRUE, 
		ModuleOutput:= ModuleOutput, 
		done=> , 
		busy=> , 
		error=> );
		IF fbWrite.done THEN
			writeestablished := TRUE;
		END_IF
		
		state := 2;
		
		
	
		
		
END_CASE
END_IF
IF (readestablished AND writeestablished) THEN
	established := TRUE;
END_IF
IF fbWrite.error OR fbRead.error THEN 
	error := TRUE;
END_IF

END_FUNCTION_BLOCK

// ---- POUs/SkillHandle/FB_2001_doublecookie.TcPOU
FUNCTION_BLOCK FB_2001_doublecookie
VAR_INPUT
	execute: BOOL;
END_VAR
VAR
	TIMERDONE: BOOL;
END_VAR

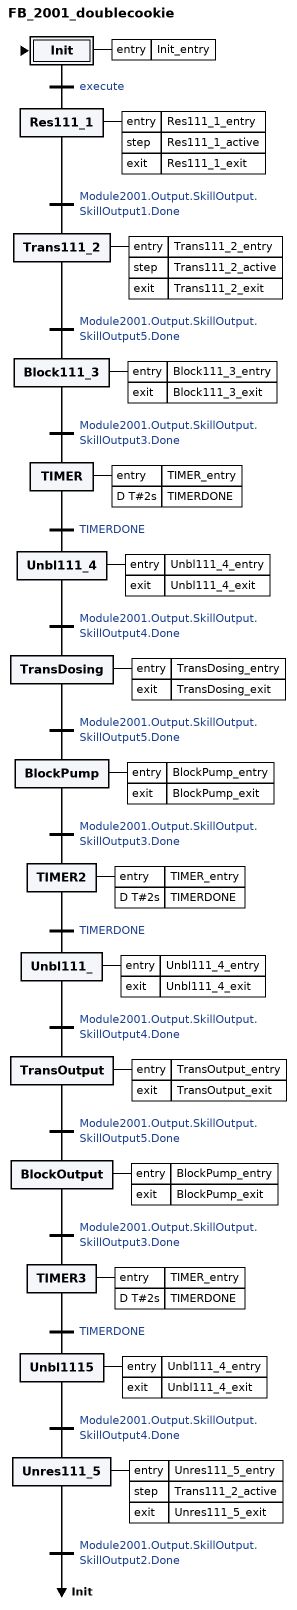
INITIAL_STEP Init:
    Init_entry(P1);  // entry action
END_STEP
TRANSITION FROM Init TO Res111_1
    := execute;
END_TRANSITION
STEP Res111_1:
    Res111_1_entry(P1);  // entry action
    Res111_1_active(N);  // step action
    Res111_1_exit(P0);  // exit action
END_STEP
TRANSITION FROM Res111_1 TO Trans111_2
    := Module2001.Output.SkillOutput.SkillOutput1.Done;
END_TRANSITION
STEP Trans111_2:
    Trans111_2_entry(P1);  // entry action
    Trans111_2_active(N);  // step action
    Trans111_2_exit(P0);  // exit action
END_STEP
TRANSITION FROM Trans111_2 TO Block111_3
    := Module2001.Output.SkillOutput.SkillOutput5.Done;
END_TRANSITION
STEP Block111_3:
    Block111_3_entry(P1);  // entry action
    Block111_3_exit(P0);  // exit action
END_STEP
TRANSITION FROM Block111_3 TO TIMER
    := Module2001.Output.SkillOutput.SkillOutput3.Done;
END_TRANSITION
STEP TIMER:
    TIMER_entry(P1);  // entry action
    TIMERDONE(D, T#2s);
END_STEP
TRANSITION FROM TIMER TO Unbl111_4
    := TIMERDONE;
END_TRANSITION
STEP Unbl111_4:
    Unbl111_4_entry(P1);  // entry action
    Unbl111_4_exit(P0);  // exit action
END_STEP
TRANSITION FROM Unbl111_4 TO TransDosing
    := Module2001.Output.SkillOutput.SkillOutput4.Done;
END_TRANSITION
STEP TransDosing:
    TransDosing_entry(P1);  // entry action
    TransDosing_exit(P0);  // exit action
END_STEP
TRANSITION FROM TransDosing TO BlockPump
    := Module2001.Output.SkillOutput.SkillOutput5.Done;
END_TRANSITION
STEP BlockPump:
    BlockPump_entry(P1);  // entry action
    BlockPump_exit(P0);  // exit action
END_STEP
TRANSITION FROM BlockPump TO TIMER2
    := Module2001.Output.SkillOutput.SkillOutput3.Done;
END_TRANSITION
STEP TIMER2:
    TIMER_entry(P1);  // entry action
    TIMERDONE(D, T#2s);
END_STEP
TRANSITION FROM TIMER2 TO Unbl111_
    := TIMERDONE;
END_TRANSITION
STEP Unbl111_:
    Unbl111_4_entry(P1);  // entry action
    Unbl111_4_exit(P0);  // exit action
END_STEP
TRANSITION FROM Unbl111_ TO TransOutput
    := Module2001.Output.SkillOutput.SkillOutput4.Done;
END_TRANSITION
STEP TransOutput:
    TransOutput_entry(P1);  // entry action
    TransOutput_exit(P0);  // exit action
END_STEP
TRANSITION FROM TransOutput TO BlockOutput
    := Module2001.Output.SkillOutput.SkillOutput5.Done;
END_TRANSITION
STEP BlockOutput:
    BlockPump_entry(P1);  // entry action
    BlockPump_exit(P0);  // exit action
END_STEP
TRANSITION FROM BlockOutput TO TIMER3
    := Module2001.Output.SkillOutput.SkillOutput3.Done;
END_TRANSITION
STEP TIMER3:
    TIMER_entry(P1);  // entry action
    TIMERDONE(D, T#2s);
END_STEP
TRANSITION FROM TIMER3 TO Unbl1115
    := TIMERDONE;
END_TRANSITION
STEP Unbl1115:
    Unbl111_4_entry(P1);  // entry action
    Unbl111_4_exit(P0);  // exit action
END_STEP
TRANSITION FROM Unbl1115 TO Unres111_5
    := Module2001.Output.SkillOutput.SkillOutput4.Done;
END_TRANSITION
STEP Unres111_5:
    Unres111_5_entry(P1);  // entry action
    Trans111_2_active(N);  // step action
    Unres111_5_exit(P0);  // exit action
END_STEP
TRANSITION FROM Unres111_5 TO Init
    := Module2001.Output.SkillOutput.SkillOutput2.Done;
END_TRANSITION

ACTION Block111_3_exit:
//BLOCKIEREN

Module2001.Input.SkillInput.SkillInput3.Execute := FALSE;
Module2001.Input.SkillInput.SkillInput3.ParameterInput.Parameterinput1.Value := 0; //TaskID
END_ACTION

ACTION TransDosing_entry:
//TRANSPORTIEREN

Module2001.Input.SkillInput.SkillInput5.Execute := TRUE;
Module2001.Input.SkillInput.SkillInput5.ParameterInput.Parameterinput1.Value := 3000; //X-Position
Module2001.Input.SkillInput.SkillInput5.ParameterInput.Parameterinput2.Value := 100;//90; //Z-Position
Module2001.Input.SkillInput.SkillInput5.ParameterInput.Parameterinput3.Value := 300; //Velocity
Module2001.Input.SkillInput.SkillInput5.ParameterInput.Parameterinput4.Value := 0; //Acceleration
END_ACTION

ACTION TransOutput_entry:
//TRANSPORTIEREN

Module2001.Input.SkillInput.SkillInput5.Execute := TRUE;
Module2001.Input.SkillInput.SkillInput5.ParameterInput.Parameterinput1.Value := 3300; //X-Position
Module2001.Input.SkillInput.SkillInput5.ParameterInput.Parameterinput2.Value := 110;//90; //Z-Position
Module2001.Input.SkillInput.SkillInput5.ParameterInput.Parameterinput3.Value := 300; //Velocity
Module2001.Input.SkillInput.SkillInput5.ParameterInput.Parameterinput4.Value := 0; //Acceleration
END_ACTION

ACTION TransOutput_exit:

Module2001.Input.SkillInput.SkillInput5.Execute := FALSE;
Module2001.Input.SkillInput.SkillInput5.ParameterInput.Parameterinput1.Value := 0; //X-Position
Module2001.Input.SkillInput.SkillInput5.ParameterInput.Parameterinput2.Value := 0; //Z-Position
Module2001.Input.SkillInput.SkillInput5.ParameterInput.Parameterinput3.Value := 0; //Velocity
Module2001.Input.SkillInput.SkillInput5.ParameterInput.Parameterinput4.Value := 0; //Acceleration
END_ACTION

ACTION Res111_1_entry:
// Reservieren entry
Module2001.Input.SkillInput.SkillInput1.Execute := TRUE;
Module2001.Input.SkillInput.SkillInput1.ParameterInput.Parameterinput1.Value := 111; //TASKID
END_ACTION

ACTION Block111_3_entry:
//BLOCKIEREN

Module2001.Input.SkillInput.SkillInput3.Execute := TRUE;
Module2001.Input.SkillInput.SkillInput3.ParameterInput.Parameterinput1.Value := 111; //TaskID
END_ACTION

ACTION Trans111_2_exit:
//TRANSPORTIEREN

Module2001.Input.SkillInput.SkillInput5.Execute := FALSE;
Module2001.Input.SkillInput.SkillInput5.ParameterInput.Parameterinput1.Value := 0; //X-Position
Module2001.Input.SkillInput.SkillInput5.ParameterInput.Parameterinput2.Value := 0; //Z-Position
Module2001.Input.SkillInput.SkillInput5.ParameterInput.Parameterinput3.Value := 0; //Velocity
Module2001.Input.SkillInput.SkillInput5.ParameterInput.Parameterinput4.Value := 0; //Acceleration
END_ACTION

ACTION Unbl111_4_exit:
//unBLOCKIEREN

Module2001.Input.SkillInput.SkillInput4.Execute := FALSE; 
Module2001.Input.SkillInput.SkillInput4.ParameterInput.Parameterinput1.Value := 000; //TaskID
END_ACTION

ACTION Unres111_5_entry:
//unreserve
Module2001.Input.SkillInput.SkillInput2.Execute := TRUE;
Module2001.Input.SkillInput.SkillInput2.ParameterInput.Parameterinput1.Value := 111; //TaskID
END_ACTION

ACTION Trans111_2_active:

END_ACTION

ACTION Init_entry:
execute := FALSE;
END_ACTION

ACTION BlockPump_entry:
//BLOCKIEREN

Module2001.Input.SkillInput.SkillInput3.Execute := TRUE;
Module2001.Input.SkillInput.SkillInput3.ParameterInput.Parameterinput1.Value := 111; //TaskID
END_ACTION

ACTION BlockPump_exit:
//BLOCKIEREN

Module2001.Input.SkillInput.SkillInput3.Execute := FALSE;
Module2001.Input.SkillInput.SkillInput3.ParameterInput.Parameterinput1.Value := 0; //TaskID
END_ACTION

ACTION Unres111_5_exit:
//unreserve
Module2001.Input.SkillInput.SkillInput2.Execute := FALSE;
Module2001.Input.SkillInput.SkillInput2.ParameterInput.Parameterinput1.Value := 0; //TaskID
END_ACTION

ACTION Trans111_2_entry:
//TRANSPORTIEREN

Module2001.Input.SkillInput.SkillInput5.Execute := TRUE;
Module2001.Input.SkillInput.SkillInput5.ParameterInput.Parameterinput1.Value := 2500; //X-Position
Module2001.Input.SkillInput.SkillInput5.ParameterInput.Parameterinput2.Value := 100;//90; //Z-Position
Module2001.Input.SkillInput.SkillInput5.ParameterInput.Parameterinput3.Value := 300; //Velocity
Module2001.Input.SkillInput.SkillInput5.ParameterInput.Parameterinput4.Value := 0; //Acceleration
END_ACTION

ACTION Res111_1_exit:
// Reservieren entry
Module2001.Input.SkillInput.SkillInput1.Execute := FALSE;
Module2001.Input.SkillInput.SkillInput1.ParameterInput.Parameterinput1.Value := 0; //TASKID
END_ACTION

ACTION TransDosing_exit:
//TRANSPORTIEREN

Module2001.Input.SkillInput.SkillInput5.Execute := FALSE;
Module2001.Input.SkillInput.SkillInput5.ParameterInput.Parameterinput1.Value := 0; //X-Position
Module2001.Input.SkillInput.SkillInput5.ParameterInput.Parameterinput2.Value := 0; //Z-Position
Module2001.Input.SkillInput.SkillInput5.ParameterInput.Parameterinput3.Value := 0; //Velocity
Module2001.Input.SkillInput.SkillInput5.ParameterInput.Parameterinput4.Value := 0; //Acceleration
END_ACTION

ACTION Res111_1_active:

END_ACTION

ACTION Unbl111_4_entry:
//unBLOCKIEREN

Module2001.Input.SkillInput.SkillInput4.Execute := TRUE; //FALSE weil timer
Module2001.Input.SkillInput.SkillInput4.ParameterInput.Parameterinput1.Value := 111; //TaskID
END_ACTION

ACTION TIMER_entry:
TIMERDONE := FALSE;
END_ACTION

END_FUNCTION_BLOCK
